TYPE ST_OutputsProfileCheck :
STRUCT

END_STRUCT
END_TYPE

(* stored: Version 1.1.0.1, ProductVersion 3.1.4024.9
   DUT ST_OutputsProfileCheck: Id {df3ec17a-7989-412f-b601-298f90cc26e3} *)
